INTERFACE I_StringLookupLREAL EXTENDS I_Fallible


METHOD Lookup
VAR_INPUT
    StringToLookup : T_MaxString;
    Result : I_QuantityLREALPublic;
END_VAR
END_METHOD

END_INTERFACE

(* stored: Version 1.1.0.1
   Itf I_StringLookupLREAL: Id {674c74e5-87a8-4d86-bcac-d267f06a9630}
   Method Lookup: Id {cec974d9-256d-43bf-826a-e26013831226} *)
